FUNCTION_BLOCK "FbDriverRTC"
TITLE = 'Блок чтения часов реального времени.'

{ S7_read_back := 'true' ;
  S7_blockview := 'big'  }

AUTHOR  : VA
FAMILY  : LIB_PLC
VERSION : '3.2'

VAR_INPUT // Входные переменные, сохраняемые.
Reset       :BOOL := FALSE; // Сброс при перезагрузке.
END_VAR

VAR_OUTPUT // Выходные переменные, сохраняемые.
Year        :INT  := 0    ; // Текущее время- Год 20xx.
Month       :INT  := 0    ; // Текущее время- Месяц 1...12.
Day         :INT  := 0    ; // Текущее время- День 1...31.
Hour        :INT  := 0    ; // Текущее время- Час 0...23.
Minute      :INT  := 0    ; // Текущее время- Минута 0...59.
Second      :INT  := 0    ; // Текущее время- Секунда 0...59.
Millisecond :INT  := 0    ; // Текущее время- Миллисекунды 0...999.
Weekday     :INT  := 0    ; // Текущее время- День недели 1...7.
Ts_ms       :DINT := 0    ; // Шаг дискретизации по времени [мс].
Ts          :REAL := 0.0  ; // Шаг дискретизации по времени [с].
Ts_max      :DINT := 0    ; // Максимальное время скана [мс].
Blink1s     :BOOL := FALSE; // Моргание 500ms ON + 500ms OFF.
END_VAR

VAR // Внутренние переменные, сохраняемые.
// Переменные для часов реального времени.
DateAndTime:DATE_AND_TIME:=DT#1999-12-31-23:59:59.999; // Дата и время 64бит.
StructDateAndTime AT DateAndTime: STRUCT // Представить 64 бит DATE_AND_TIME как восемь BYTE
ArrayByte:ARRAY[0..7] OF BYTE; // Массив из 8 байт.
// ArrayByte[0] Год в формате BCD.
// ArrayByte[1] Месяц в формате BCD.
// ArrayByte[2] День в формате BCD.
// ArrayByte[3] Час в формате BCD.
// ArrayByte[4] Минута в формате BCD.
// ArrayByte[5] Секунда в формате BCD.
// ArrayByte[6] Милисекунда в формате BCD.
// ArrayByte[7] Милисекунды и день недели в формате BCD.
END_STRUCT;
Time_ms_previous :DINT := 0; // RTC предидущее значение 0...59999ms.
END_VAR

VAR_TEMP  // Временные переменные, не сохраняемые.
ErrorCode       :INT ; // Код ошики SFC должен быть 0.
TmpBYTE         :BYTE; // Временная переменная.
ms_x10          :BYTE; // Временная переменная 1.
ms_x100         :BYTE; // Временная переменная 2.
ms_x1           :BYTE; // Временная переменная 3.
Time_ms_current :DINT; // RTC 0...59999ms.
END_VAR

BEGIN

// Блок чтения часов реального времени.
//         DbDriverRTC
//     +-----------------+
//     |   FbDriverRTC   |
//  ->-|Reset        Year|->-
//     |            Month|->-
//     |              Day|->-
//     |             Hour|->-
//     |          Minutes|->-
//     |          Seconds|->-
//     |      Millisecond|->-
//     |          Weekday|->-
//     |            Ts_ms|->-
//     |               Ts|->-
//     |           Ts_max|->-
//     |          Blink1s|->-
//     +-----------------+

// Чтение RTC.
ErrorCode := READ_CLK(CDT:=DateAndTime); // SFC1();
IF (ErrorCode = 0) THEN

// Расшифровка BCD формата времени- год.
Year := 2000 + BCD_TO_INT(StructDateAndTime.ArrayByte[0]);

// Расшифровка BCD формата времени- месяц.
Month := BCD_TO_INT(StructDateAndTime.ArrayByte[1]);

// Расшифровка BCD формата времени- день.
Day := BCD_TO_INT(StructDateAndTime.ArrayByte[2]);

// Расшифровка BCD формата времени- час.
Hour := BCD_TO_INT(StructDateAndTime.ArrayByte[3]);

// Расшифровка BCD формата времени- минута.
Minute := BCD_TO_INT(StructDateAndTime.ArrayByte[4]);

// Расшифровка BCD формата времени- секунда.
Second := BCD_TO_INT(StructDateAndTime.ArrayByte[5]);

// Расшифровка BCD формата времени- миллисекунда.
ms_x10  := StructDateAndTime.ArrayByte[6] AND 2#0000_1111; // ms x10
ms_x100 := ROR(IN:=StructDateAndTime.ArrayByte[6] AND 2#1111_0000,N:=4); // ms x100
ms_x1   := ROR(IN:=StructDateAndTime.ArrayByte[7] AND 2#1111_0000,N:=4); // ms x1
Millisecond := BYTE_TO_INT(ms_x100)*100 + BYTE_TO_INT(ms_x10)*10 + BYTE_TO_INT(ms_x1);

// Расшифровка BCD формата времени- день недели.
Weekday := BYTE_TO_INT(StructDateAndTime.ArrayByte[7] AND 2#0000_1111);

ELSE
Year        := 0;
Month       := 0;
Day         := 0;
Hour        := 0;
Minute      := 0;
Second      := 0;
Millisecond := 0;
Weekday     := 0;
END_IF;

//--------------------------------------------------------------------------------------------

// Моргание 500ms ON + 500ms OFF.
Blink1s := Millisecond <= 499;

//--------------------------------------------------------------------------------------------

// Расчет времени скана ПЛК с точки зрения RTC.
// Может быть полезна для OB1 в S7-1200 и для OB1 в CFC PCS7.

// RTC 0...59999ms
Time_ms_current := (INT_TO_DINT(Second) * 1000) + INT_TO_DINT(Millisecond);

// Инициализируем время при перезагрузке.
IF (Reset) THEN
Time_ms_previous := Time_ms_current;
END_IF;

// Разность времени с учетом переполнения.
IF (Time_ms_current >= Time_ms_previous) THEN
Ts_ms := Time_ms_current - Time_ms_previous;
// Ts_ms = 7 - 2 = 5 ms
// 0
// 1
// 2 <- Time_ms_previous
// 3
// 4
// 5
// 6
// 7 <- Time_ms_current
// 8
// 9
ELSE
Ts_ms := (60000 - Time_ms_previous) + Time_ms_current;
// Ts_ms = (60000 - 59997) + 2 = 5 ms
// 59995
// 59996
// 59997 <- Time_ms_previous
// 59998
// 59999
// 0
// 1
// 2 <- Time_ms_current
// 3
// 4
END_IF;

// Запомнить предидущее время.
Time_ms_previous := Time_ms_current;

// Время скана не может быть больше 1000ms
// Защита на случай если ПЛК переведут в стоп на длительное время.
// Защита от внезапной корректировки времени RTC.
// Защита от неверных входных данных.
IF ((Ts_ms >= 1000) OR (Ts_ms < 0)) THEN
Ts_ms := 0;
END_IF;

// Шаг дискретизации по времени [с].
Ts := DINT_TO_REAL(Ts_ms) * 0.001;

//--------------------------------------------------------------------------------------------

// Максимальное время скана [мс].
IF (Ts_ms >= Ts_max) THEN
Ts_max := Ts_ms;
END_IF;

IF (Reset) THEN
Ts_max := 0;
END_IF;

//--------------------------------------------------------------------------------------------

// @COPYLEFT ALL WRONGS RESERVED :)
// Author: VA
// Contacts: DIY.PLC.314@gmail.com
// Date start LIB_PLC: 2014
// License: GNU GPL-2.0-or-later
// https://www.gnu.org/licenses/old-licenses/gpl-2.0.html
// https://www.youtube.com/watch?v=n1F_MfLRlX0
// https://www.youtube.com/@DIY_PLC
// https://github.com/DIYPLC/LIB_PLC
// https://oshwlab.com/diy.plc.314/PLC_HW1_SW1
// https://3dtoday.ru/3d-models/mechanical-parts/body/korpus-na-din-reiku
// https://t.me/DIY_PLC
// https://drive.google.com/drive/folders/16GDX0i07rwDrl_oPzL-lQAqMiAz3ouJV?usp=sharing

END_FUNCTION_BLOCK
